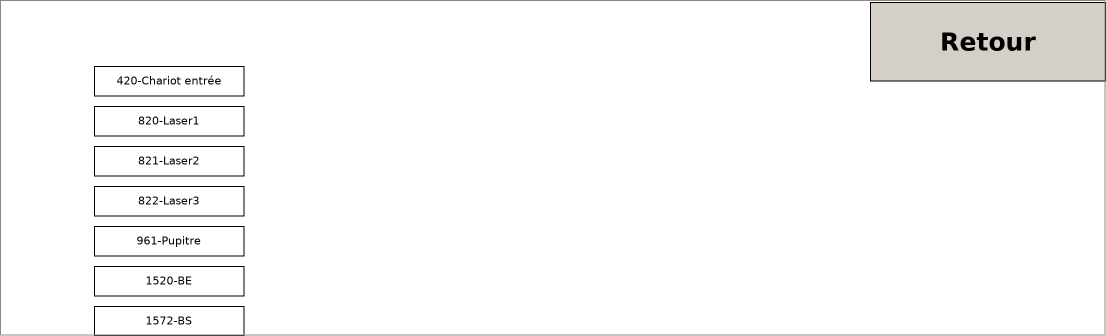
VISUALIZATION Selection_Rep  // 1106x336
    Rectangle (94,106 150x30), "820-Laser1"
        OnMouseClick: execute { Forcage_Rep.Num_Rep_Selectionne_pr_Forcage:=2; }
        OnMouseUp: change screen: VisuForce
    Rectangle (94,146 150x30), "821-Laser2"
        OnMouseClick: execute { Forcage_Rep.Num_Rep_Selectionne_pr_Forcage:=3; }
        OnMouseUp: change screen: VisuForce
    Rectangle (94,186 150x30), "822-Laser3"
        OnMouseClick: execute { Forcage_Rep.Num_Rep_Selectionne_pr_Forcage:=4; }
        OnMouseUp: change screen: VisuForce
    Rectangle (94,66 150x30), "420-Chariot entrée"
        OnMouseClick: execute { Forcage_Rep.Num_Rep_Selectionne_pr_Forcage:=1; }
        OnMouseUp: change screen: VisuForce
    Rectangle (94,226 150x30), "961-Pupitre"
        OnMouseClick: execute { Forcage_Rep.Num_Rep_Selectionne_pr_Forcage:=5; }
        OnMouseUp: change screen: VisuForce
    Rectangle (94,266 150x30), "1520-BE"
        OnMouseClick: execute { Forcage_Rep.Num_Rep_Selectionne_pr_Forcage:=6; }
        OnMouseUp: change screen: VisuForce
    Rectangle (94,306 150x30), "1572-BS"
        OnMouseClick: execute { Forcage_Rep.Num_Rep_Selectionne_pr_Forcage:=7; }
        OnMouseUp: change screen: VisuForce
    Rectangle (870,2 236x79), "Retour"
        OnMouseClick: change screen: MenuPrincipal
        OnMouseClick: execute { Forcage_Rep.Num_Rep_Selectionne_pr_Forcage:=0; }
END_VISUALIZATION

(* stored: Version 1.1.0.1
   Visu Selection_Rep: Id {2c843dac-a0eb-4825-a54e-f2e1da563584} *)
